FUNCTION_BLOCK VIEW_HMI (* HMI for testing Views with Position and Color *)
  (* Standard: 61499-1; ApplicationDomain: MVA_CDA; Function: HMI *)
  (* Version 0.0, 2001-03-04, JHC, Rockwell Automation *)
  (* Compiler header: package fb.rt.omac; import fb.rt.hmi.*; *)
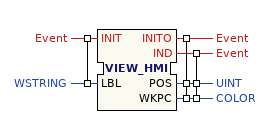
  EVENT_INPUT
    INIT WITH LBL;
  END_EVENT
  EVENT_OUTPUT
    INITO WITH POS, WKPC;
    IND WITH POS, WKPC;
  END_EVENT
  VAR_INPUT
    LBL : WSTRING;
  END_VAR
  VAR_OUTPUT
    POS : UINT;
    WKPC : COLOR;
  END_VAR
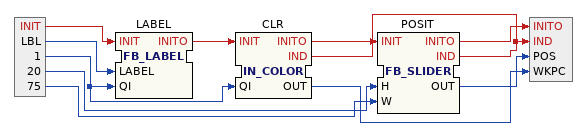
  FBS
    LABEL : FB_LABEL;
    CLR : IN_COLOR;
    POSIT : FB_SLIDER;
  END_FBS
  EVENT_CONNECTIONS
    INIT TO LABEL.INIT;
    LABEL.INITO TO CLR.INIT;
    CLR.INITO TO POSIT.INIT;
    POSIT.INITO TO INITO;
    CLR.IND TO IND;
    POSIT.IND TO IND;
  END_CONNECTIONS
  DATA_CONNECTIONS
    LBL TO LABEL.LABEL;
    CLR.OUT TO WKPC;
    POSIT.OUT TO POS;
    1 TO LABEL.QI;
    1 TO CLR.QI;
    20 TO POSIT.H;
    75 TO POSIT.W;
  END_CONNECTIONS
END_FUNCTION_BLOCK
